Fanuc TP program (LS listing): up223.ls

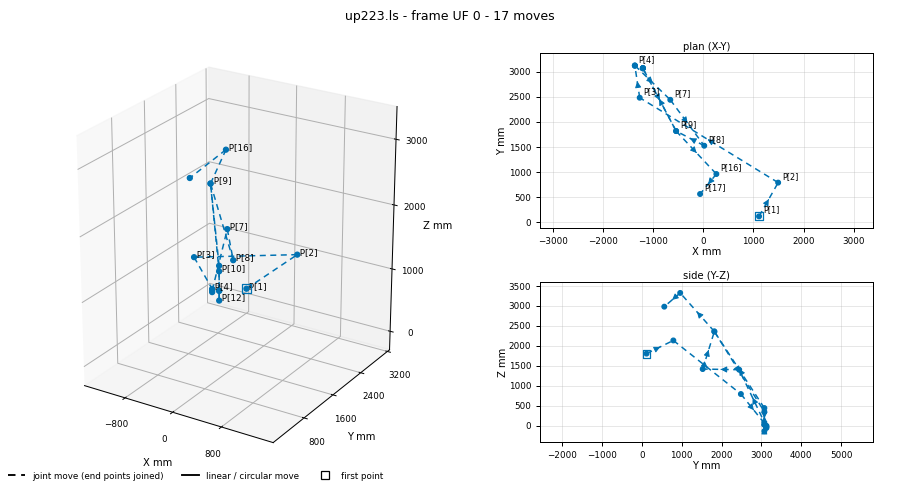
[picture p0: tool path of up223.ls in frame UF 0, 17 of 17 moves have a stored position in this frame; points joined in program order, loops and branches not executed]
/PROG  UP223
/ATTR
OWNER		= MNEDITOR;
COMMENT		= "Dejar en ST1600";
PROG_SIZE	= 9152;
CREATE		= DATE 23-07-09  TIME 16:00:56;
MODIFIED	= DATE 23-07-09  TIME 16:00:58;
FILE_NAME	= UP023;
VERSION		= 0;
LINE_COUNT	= 35;
MEMORY_SIZE	= 15604;
PROTECT		= READ_WRITE;
TCD:  STACK_SIZE	= 500,
      TASK_PRIORITY	= 50,
      TIME_SLICE	= 0,
      BUSY_LAMP_OFF	= 0,
      ABORT_REQUEST	= 0,
      PAUSE_REQUEST	= 0;
DEFAULT_GROUP	= 1,1,1,1,*;
CONTROL_CODE	= 00000000 00000000;
/APPL
/MN
   1:  UFRAME_NUM=0 ;
   2:  UTOOL_NUM=2 ;
   3:  PAYLOAD[3] ;
   4:  !Apagar Perfil Lib. 73 vs ST1600 ;
   5:  !Apagar Perfil Lib. 72 vs ST1600 ;
   6:  !Encender Anticol. 1 vs 1600R01 ;
   7:  !Encender Anticol. 7 vs 1610R01 ;
   8:J P[1] 100% CNT0 ACC100 TB    .10sec,P-SPS    ;
      1:  TC_ONLINE (ON) ;
      2:  DO[23]=(OFF) ;
      3:  TIMER[5]=RESET ;
      4:  TIMER[5]=START ;
      5:  CALL MAKRO050    ;
      6:  !Lib. de Herramientas ;
      7:  DO[80]=ON ;
      8:  DO[79]=ON ;
      9:  DO[78]=OFF ;
     10:  DO[77]=OFF ;
     11:  DO[76]=ON ;
     12:  DO[75]=OFF ;
     13:  DO[74]=OFF ;
     14:  DO[73]=ON ;
     15:  DO[72]=ON ;
     16:  DO[70]=OFF ;
     17:  DO[69]=OFF ;
     18:  DO[68]=OFF ;
     19:  DO[67]=OFF ;
     20:  !Lib. de Anticolisiones ;
     21:  DO[41]=ON ;
     22:  DO[42]=ON ;
     23:  DO[43]=ON ;
     24:  DO[44]=ON ;
     25:  DO[45]=ON ;
     26:  DO[46]=ON ;
     27:  DO[47]=ON ;
     28:  DO[48]=ON ;
     29:  !Apagar Posicion Base ;
     30:  DO[15]=OFF ;
     31:  !Roboter en Trayectoria ;
     32:  DO[16]=ON ;
     33:  WAIT (DI[57] AND !DI[58] AND DI[59] AND !DI[60] AND DI[73] AND DI[72])    ;
     34:  DO[73]=OFF ;
     35:  DO[72]=OFF ;
     36:  DO[81]=ON ;
     37:  DO[87]=ON ;
     38:  CALL MAKRO020    ;
     39:  WAIT (DI[23])    ;
     40:  DO[23]=ON ;
     41:  !Marca Usuario ST1600 S/Pieza 1 ;
     42:  !M[19] = (DI[59] AND !DI[60]) ;
     43:  !Marca Usuario ST1600 S/Pieza 2 ;
     44:  !M[21] = (DI[57] AND !DI[58]) ;
     45:  !Marca de Usuario Suma de Anticol ;
     46:  !M[22] = (DI[41] AND DI[47]) ;
     47:  !Marca de Usuario Estado de Garra ;
     48:  !M[23] = (M[32] AND M[38]]) ;
     49:  !Marca de Usuario Estado de Garra ;
     50:  !M[26] = (M[39] AND M[41] AND M[4 ;
     51:  TC_ONLINE (DI[72] AND DI[73] AND M[1] AND M[19] AND M[21] AND M[22] AND M[23] AND M[26] AND M[30] AND M[33] AND M[36]) ;
       ------ ;
   9:J P[2] 100% CNT100 ACC100 TB   0.00sec,P-SPS    ;
      1:  TC_ONLINE (DI[72] AND DI[73] AND M[1] AND M[19] AND M[21] AND M[22] AND M[23] AND M[26] AND M[30] AND M[33] AND M[36]) ;
       ------ ;
  10:J P[3] 100% CNT100 ACC100 TB   0.00sec,P-SPS    ;
      1:  TC_ONLINE (DI[72] AND DI[73] AND M[1] AND M[19] AND M[21] AND M[22] AND M[23] AND M[26] AND M[30] AND M[33] AND M[36]) ;
       ------ ;
  11:J P[4] 100% CNT0 ACC100 TB    .10sec,P-SPS    ;
      1:  TC_ONLINE (ON) ;
      2:  DO[23]=(OFF) ;
      3:  F[2]=(ON) ;
      4:  CALL MAKRO343    ;
      5:  WAIT (M[34])    ;
      6:  WAIT (DI[23])    ;
      7:  DO[23]=(ON) ;
      8:  TC_ONLINE (DI[72] AND DI[73] AND M[1] AND M[21] AND M[22] AND M[23] AND M[26] AND M[30] AND M[34] AND M[36]) ;
       ------ ;
  12:  !En Posicion ST1600 ;
  13:  !Dejar Pieza 1 en ST1600 ;
  14:  !Fin de Trabajo 4 ;
  15:L P[5] 1500mm/sec CNT0 ACC100 TB    .10sec,P-SPS    ;
      1:  TC_ONLINE (ON) ;
      2:  DO[23]=OFF ;
      3:  WAIT ((!DI[59] AND DI[60]) OR DI[15])    ;
      4:  DO[70]=ON ;
      5:  CALL MAKRO004    ;
      6:  WAIT (DI[71])    ;
      7:  DO[70]=OFF ;
      8:  F[3]=(ON) ;
      9:  CALL MAKRO342    ;
     10:  CALL MAKRO340    ;
     11:  WAIT (M[35])    ;
     12:  WAIT (DI[23])    ;
     13:  DO[23]=(ON) ;
     14:  !Marca Usuario ST1600 C/Pieza 1 ;
     15:  !M[18] = (!DI[59] AND DI[60]) ;
     16:  TC_ONLINE (DI[71] AND DI[73] AND M[18] AND M[21] AND M[22] AND M[23] AND M[26] AND M[30] AND M[34] AND M[35]) ;
       ------ ;
  16:L P[6] 2000mm/sec CNT0 ACC100 TB    .10sec,P-SPS    ;
      1:  TC_ONLINE (ON) ;
      2:  DO[23]=(OFF) ;
      3:  WAIT (!DI[59] AND DI[60] AND M[5])    ;
      4:  WAIT (DI[23])    ;
      5:  DO[23]=(ON) ;
      6:  TC_ONLINE (DI[71] AND DI[73] AND M[5] AND M[18] AND M[21] AND M[22] AND M[23] AND M[26] AND M[30] AND M[34] AND M[35]) ;
       ------ ;
  17:  UTOOL_NUM=1 ;
  18:J P[7] 100% CNT100 ACC100 TB   0.00sec,P-SPS    ;
      1:  TC_ONLINE (DI[71] AND DI[73] AND M[5] AND M[18] AND M[21] AND M[22] AND M[23] AND M[26] AND M[30] AND M[34] AND M[35]) ;
       ------ ;
  19:J P[8] 100% CNT0 ACC100 TB    .10sec,P-SPS    ;
      1:  TC_ONLINE (ON) ;
      2:  DO[23]=(OFF) ;
      3:  DO[69]=(ON) ;
      4:  WAIT (DI[69])    ;
      5:  DO[69]=(OFF) ;
      6:  WAIT (DI[23])    ;
      7:  DO[23]=(ON) ;
      8:  TC_ONLINE (DI[69] AND DI[73] AND M[5] AND M[18] AND M[21] AND M[22] AND M[23] AND M[26] AND M[30] AND M[34] AND M[35]) ;
       ------ ;
  20:J P[9] 100% CNT100 ACC100 TB   0.00sec,P-SPS    ;
      1:  TC_ONLINE (DI[69] AND DI[73] AND M[5] AND M[18] AND M[21] AND M[22] AND M[23] AND M[26] AND M[30] AND M[34] AND M[35]) ;
       ------ ;
  21:J P[10] 100% CNT100 ACC100 TB   0.00sec,P-SPS    ;
      1:  TC_ONLINE (DI[69] AND DI[73] AND M[5] AND M[18] AND M[21] AND M[22] AND M[23] AND M[26] AND M[30] AND M[34] AND M[35]) ;
       ------ ;
  22:J P[11] 100% CNT0 ACC100 TB    .10sec,P-SPS    ;
      1:  TC_ONLINE (ON) ;
      2:  DO[23]=(OFF) ;
      3:  F[5]=(ON) ;
      4:  F[6]=(ON) ;
      5:  F[7]=(ON) ;
      6:  CALL MAKRO343    ;
      7:  WAIT (M[40] AND M[42] AND M[44])    ;
      8:  WAIT (DI[23])    ;
      9:  DO[23]=(ON) ;
     10:  !Marca de Usuario Estado de Garra ;
     11:  !M[25] = (M[40] AND M[42] AND M[4 ;
     12:  TC_ONLINE (DI[69] AND DI[73] AND M[5] AND M[18] AND M[22] AND M[23] AND M[25] AND M[30] AND M[34] AND M[35]) ;
       ------ ;
  23:  !En Posicion ST1600 ;
  24:  !Dejar Pieza 2 en ST1600 ;
  25:  !Fin de Trabajo 5 ;
  26:L P[12] 1500mm/sec CNT0 ACC100 TB    .10sec,P-SPS    ;
      1:  TC_ONLINE (ON) ;
      2:  DO[23]=OFF ;
      3:  WAIT ((!DI[57] AND DI[58]) OR DI[15])    ;
      4:  DO[67]=ON ;
      5:  DO[68]=ON ;
      6:  CALL MAKRO005    ;
      7:  WAIT (DI[68])    ;
      8:  DO[68]=OFF ;
      9:  DO[67]=OFF ;
     10:  F[1]=(ON) ;
     11:  F[4]=(ON) ;
     12:  CALL MAKRO342    ;
     13:  CALL MAKRO340    ;
     14:  WAIT (M[31] AND M[37])    ;
     15:  WAIT (DI[23])    ;
     16:  DO[23]=(ON) ;
     17:  !Marca de Usuario Estado de Garra ;
     18:  !M[24] = (M[31] AND M[37]) ;
     19:  !Marca Usuario ST1600 C/Pieza 2 ;
     20:  !M[20] = (!DI[57] AND DI[58]) ;
     21:  TC_ONLINE (DI[68] AND DI[73] AND M[18] AND M[20] AND M[22] AND M[24] AND M[25] AND M[30] AND M[34] AND M[35]) ;
       ------ ;
  27:L P[13] 2000mm/sec CNT100 ACC100 TB   0.00sec,P-SPS    ;
      1:  TC_ONLINE (DI[68] AND DI[73] AND M[2] AND M[18] AND M[20] AND M[22] AND M[24] AND M[25] AND M[30] AND M[34] AND M[35]) ;
       ------ ;
  28:J P[14] 100% CNT100 ACC100 TB   0.00sec,P-SPS    ;
      1:  TC_ONLINE (DI[68] AND DI[73] AND M[2] AND M[18] AND M[20] AND M[22] AND M[24] AND M[25] AND M[30] AND M[34] AND M[35]) ;
       ------ ;
  29:J P[15] 100% CNT100 ACC100 TB   0.00sec,P-SPS    ;
      1:  TC_ONLINE (DI[68] AND DI[73] AND M[2] AND M[18] AND M[20] AND M[22] AND M[24] AND M[25] AND M[30] AND M[34] AND M[35]) ;
       ------ ;
  30:J P[16] 100% CNT100 ACC100 TB   0.00sec,P-SPS    ;
      1:  TC_ONLINE (DI[68] AND DI[73] AND M[2] AND M[18] AND M[20] AND M[22] AND M[24] AND M[25] AND M[30] AND M[34] AND M[35]) ;
       ------ ;
  31:  !Encender Perfil Lib 73 vs ST1600 ;
  32:  !Encender Perfil Lib 72 vs ST1600 ;
  33:  !Apagar Anticol. 1 vs 1600R01 ;
  34:  !Apagar Anticol. 7 vs 1610R01 ;
  35:J P[17] 100% CNT0 ACC100 TB    .10sec,P-SPS    ;
      1:  TC_ONLINE (ON) ;
      2:  DO[23]=OFF ;
      3:  TIMER[5]=STOP ;
      4:  F[2]=(ON) ;
      5:  F[5]=(ON) ;
      6:  F[6]=(ON) ;
      7:  F[7]=(ON) ;
      8:  CALL MAKRO342    ;
      9:  CALL MAKRO340    ;
     10:  WAIT (M[33] AND M[39] AND M[41] AND M[43])    ;
     11:  DO[41]=ON ;
     12:  DO[47]=ON ;
     13:  DO[73]=ON ;
     14:  DO[72]=ON ;
     15:  WAIT (DI[23])    ;
     16:  DO[23]=ON ;
     17:  TC_ONLINE (M[2] AND M[30] AND M[31] AND M[33] AND M[35] AND M[37] AND M[39] AND M[41] AND M[43]) ;
       ------ ;
/POS
P[1]{
   GP1:
	UF : 0, UT : 2,		CONFIG : 'N U T, 0, 0, 0',
	X =  1111.865  mm,	Y =   118.787  mm,	Z =  1806.347  mm,
	W =   -70.737 deg,	P =    11.951 deg,	R =   -35.487 deg
   GP2:
	UF : 0, UT : 2,
	J1=     0.000  mm
   GP3:
	UF : 0, UT : 2,
	J1=     0.000  mm
   GP4:
	UF : 0, UT : 2,
	J1=     0.000  mm
};
P[2]{
   GP1:
	UF : 0, UT : 2,		CONFIG : 'N U T, 0, 0, 0',
	X =  1492.784  mm,	Y =   791.366  mm,	Z =  2136.380  mm,
	W =   -74.744 deg,	P =    11.683 deg,	R =   -19.804 deg
   GP2:
	UF : 0, UT : 2,
	J1=     0.000  mm
   GP3:
	UF : 0, UT : 2,
	J1=     0.000  mm
   GP4:
	UF : 0, UT : 2,
	J1=     0.000  mm
};
P[3]{
   GP1:
	UF : 0, UT : 2,		CONFIG : 'N U T, 0, 0, 0',
	X = -1267.629  mm,	Y =  2484.028  mm,	Z =   793.110  mm,
	W =    90.000 deg,	P =    55.000 deg,	R =   143.543 deg
   GP2:
	UF : 0, UT : 2,
	J1=     0.000  mm
   GP3:
	UF : 0, UT : 2,
	J1=     0.000  mm
   GP4:
	UF : 0, UT : 2,
	J1=     0.000  mm
};
P[4]{
   GP1:
	UF : 0, UT : 2,		CONFIG : 'N U T, 0, 0, 0',
	X = -1364.414  mm,	Y =  3123.377  mm,	Z =    -2.798  mm,
	W =    59.389 deg,	P =    89.796 deg,	R =   105.320 deg
   GP2:
	UF : 0, UT : 2,
	J1=     0.000  mm
   GP3:
	UF : 0, UT : 2,
	J1=     0.000  mm
   GP4:
	UF : 0, UT : 2,
	J1=     0.000  mm
};
P[5]{
   GP1:
	UF : 0, UT : 2,		CONFIG : 'N U T, 0, 0, 0',
	X = -1364.461  mm,	Y =  3123.562  mm,	Z =   -57.299  mm,
	W =    59.392 deg,	P =    89.796 deg,	R =   105.323 deg
   GP2:
	UF : 0, UT : 2,
	J1=     0.000  mm
   GP3:
	UF : 0, UT : 2,
	J1=     0.000  mm
   GP4:
	UF : 0, UT : 2,
	J1=     0.000  mm
};
P[6]{
   GP1:
	UF : 0, UT : 2,		CONFIG : 'N U T, 0, 0, 0',
	X = -1363.757  mm,	Y =  3125.704  mm,	Z =   -27.132  mm,
	W =    59.233 deg,	P =    89.796 deg,	R =   105.164 deg
   GP2:
	UF : 0, UT : 2,
	J1=     0.000  mm
   GP3:
	UF : 0, UT : 2,
	J1=     0.000  mm
   GP4:
	UF : 0, UT : 2,
	J1=     0.000  mm
};
P[7]{
   GP1:
	UF : 0, UT : 1,		CONFIG : 'N U T, 0, 0, 0',
	X =  -657.589  mm,	Y =  2442.038  mm,	Z =  1402.206  mm,
	W =   -44.819 deg,	P =      .153 deg,	R =    45.932 deg
   GP2:
	UF : 0, UT : 1,
	J1=     0.000  mm
   GP3:
	UF : 0, UT : 1,
	J1=     0.000  mm
   GP4:
	UF : 0, UT : 1,
	J1=     0.000  mm
};
P[8]{
   GP1:
	UF : 0, UT : 1,		CONFIG : 'N U T, 0, 0, 0',
	X =    19.353  mm,	Y =  1526.865  mm,	Z =  1419.539  mm,
	W =   -10.000 deg,	P =     0.000 deg,	R =    53.543 deg
   GP2:
	UF : 0, UT : 1,
	J1=     0.000  mm
   GP3:
	UF : 0, UT : 1,
	J1=     0.000  mm
   GP4:
	UF : 0, UT : 1,
	J1=     0.000  mm
};
P[9]{
   GP1:
	UF : 0, UT : 1,		CONFIG : 'N U T, 0, 0, 0',
	X =  -541.428  mm,	Y =  1819.070  mm,	Z =  2360.446  mm,
	W =   -81.330 deg,	P =    -5.106 deg,	R =    53.050 deg
   GP2:
	UF : 0, UT : 1,
	J1=     0.000  mm
   GP3:
	UF : 0, UT : 1,
	J1=     0.000  mm
   GP4:
	UF : 0, UT : 1,
	J1=     0.000  mm
};
P[10]{
   GP1:
	UF : 0, UT : 1,		CONFIG : 'N U T, 0, 0, 0',
	X = -1205.386  mm,	Y =  3072.959  mm,	Z =   348.202  mm,
	W =  -133.491 deg,	P =    89.681 deg,	R =    92.122 deg
   GP2:
	UF : 0, UT : 1,
	J1=     0.000  mm
   GP3:
	UF : 0, UT : 1,
	J1=     0.000  mm
   GP4:
	UF : 0, UT : 1,
	J1=     0.000  mm
};
P[11]{
   GP1:
	UF : 0, UT : 1,		CONFIG : 'N U T, 0, 0, 0',
	X = -1204.866  mm,	Y =  3071.746  mm,	Z =    25.723  mm,
	W =  -172.540 deg,	P =    88.689 deg,	R =    52.786 deg
   GP2:
	UF : 0, UT : 1,
	J1=     0.000  mm
   GP3:
	UF : 0, UT : 1,
	J1=     0.000  mm
   GP4:
	UF : 0, UT : 1,
	J1=     0.000  mm
};
P[12]{
   GP1:
	UF : 0, UT : 1,		CONFIG : 'N U T, 0, 0, 0',
	X = -1204.905  mm,	Y =  3071.697  mm,	Z =  -138.503  mm,
	W =  -167.717 deg,	P =    88.670 deg,	R =    57.610 deg
   GP2:
	UF : 0, UT : 1,
	J1=     0.000  mm
   GP3:
	UF : 0, UT : 1,
	J1=     0.000  mm
   GP4:
	UF : 0, UT : 1,
	J1=     0.000  mm
};
P[13]{
   GP1:
	UF : 0, UT : 1,		CONFIG : 'N U T, 0, 0, 0',
	X = -1204.866  mm,	Y =  3071.746  mm,	Z =    25.723  mm,
	W =  -172.540 deg,	P =    88.689 deg,	R =    52.786 deg
   GP2:
	UF : 0, UT : 1,
	J1=     0.000  mm
   GP3:
	UF : 0, UT : 1,
	J1=     0.000  mm
   GP4:
	UF : 0, UT : 1,
	J1=     0.000  mm
};
P[14]{
   GP1:
	UF : 0, UT : 1,		CONFIG : 'N U T, 0, 0, 0',
	X = -1204.417  mm,	Y =  3072.711  mm,	Z =   441.462  mm,
	W =   -38.476 deg,	P =    89.769 deg,	R =  -172.579 deg
   GP2:
	UF : 0, UT : 1,
	J1=     0.000  mm
   GP3:
	UF : 0, UT : 1,
	J1=     0.000  mm
   GP4:
	UF : 0, UT : 1,
	J1=     0.000  mm
};
P[15]{
   GP1:
	UF : 0, UT : 1,		CONFIG : 'N U T, 0, 0, 0',
	X =  -541.433  mm,	Y =  1819.071  mm,	Z =  2360.436  mm,
	W =   -81.330 deg,	P =    -5.106 deg,	R =    53.050 deg
   GP2:
	UF : 0, UT : 1,
	J1=     0.000  mm
   GP3:
	UF : 0, UT : 1,
	J1=     0.000  mm
   GP4:
	UF : 0, UT : 1,
	J1=     0.000  mm
};
P[16]{
   GP1:
	UF : 0, UT : 1,		CONFIG : 'N U T, 0, 0, 0',
	X =   260.814  mm,	Y =   962.826  mm,	Z =  3327.073  mm,
	W =  -122.903 deg,	P =   -14.932 deg,	R =    67.034 deg
   GP2:
	UF : 0, UT : 1,
	J1=     0.000  mm
   GP3:
	UF : 0, UT : 1,
	J1=     0.000  mm
   GP4:
	UF : 0, UT : 1,
	J1=     0.000  mm
};
P[17]{
   GP1:
	UF : 0, UT : 1,		CONFIG : 'N U T, 0, 0, 0',
	X =   -63.679  mm,	Y =   564.245  mm,	Z =  2983.021  mm,
	W =  -122.362 deg,	P =   -18.830 deg,	R =    50.373 deg
   GP2:
	UF : 0, UT : 1,
	J1=     0.000  mm
   GP3:
	UF : 0, UT : 1,
	J1=     0.000  mm
   GP4:
	UF : 0, UT : 1,
	J1=     0.000  mm
};
/END
